(* CODESYS project v35_Linux_Profinet

Project tree, tasks and I/O mapping:
  Device : CODESYS Control for Linux SL, 3S - Smart Software Solutions GmbH, version 4.5.0.0
    application Application
      libraries: Standard, * (System)
      task MainTask (cyclic, interval t#4ms, priority 1) calls PLC_PRG
      task Profinet_CommunicationTask (cyclic, interval t#10ms, priority 14) calls PN_Controller.CommCycle
      task Profinet_IOTask (cyclic, interval t#1ms, priority 1) calls nothing
      program PLC_PRG [ST]
    Ethernet : Ethernet, 3S - Smart Software Solutions GmbH, version 3.5.17.0
        settings: IPAddress = [10,10,2,5]; SubnetMask = [255,255,255,0]; GatewayAddress = [0,0,0,0]; MACAddress = [16#C4,16#00,16#AD,16#8F,16#F7,16#F8]; NetworkInterfaceName = 'X11'; NetworkInterfaceName = "X11"; SaveCommunicationSettings = FALSE
      PN_Controller : PN-Controller, 3S - Smart Software Solutions GmbH, order no. 1, version 4.2.0.0
          settings: Controller Options.IOxSSettings.PSInputDataMapped = True; Controller Options.IOxSSettings.CSOutputDataMapped = True; First IP Address = [10, 10, 2, 10]; Last IP Address = [10, 10, 2, 254]; Default Subnet Mask = [255, 255, 255, 0]; Default Gateway Address = [0, 0, 0, 0]; PDPortDataCheck.PeerStationName = ''
        RIO_Panel1A : 750-375 V02.07.xx (FW 10), WAGO Kontakttechnik GmbH & Co. KG, order no. 750-375, version SW=V02.07.xx (10), HW=01
            settings: Slave parameters.Identification.IP address = [10,10,2,10]; Slave parameters.Identification.Subnet mask = [255,255,255,0]; Slave parameters.Identification.Default gateway = [0,0,0,0]; Slave parameters.Identification.MAC address = [16#00,16#30,16#DE,16#40,16#2C,16#5D]; Slave parameters.Identification.Station name = 'wago.remote.io.2'; Slave parameters.Reduction ratio = 4; PDPortDataCheck.PeerStationName = ''; PDPortDataCheck.PeerStationName = ''
            unmapped channels: Inputs PS, Inputs PS, Inputs PS, Inputs PS
          RIO_Panel1A_S01 : 750-496 8AI 0/4-20 mA s.e., WAGO Kontakttechnik GmbH & Co. KG, order no. 750-496, version SW=V02.07.xx (10), HW=01
              settings: Module parameters.Slot number = 1
            wago_remote_io_2_2_1 : 8AI, INT16[8] I, WAGO Kontakttechnik GmbH & Co. KG, version SW=V02.07.xx (10), HW=01
                settings: 8AI, INT16[8] I.Subslot number = 1; swapInfoInputs = [7,8]
                unmapped channels: Inputs, Inputs PS
          RIO_Panel1A_S02 : 16DO, WAGO Kontakttechnik GmbH & Co. KG, order no. 750-15xx, version SW=V02.07.xx (10), HW=01
              settings: Module parameters.Slot number = 2
            wago_remote_io_2_2_1_1 : 16DO, WAGO Kontakttechnik GmbH & Co. KG, version SW=V02.07.xx (10), HW=01
                settings: 16DO.Subslot number = 1; swapInfoOutputs = [2,2]
                unmapped channels: Digital Outputs .0 - .15, Outputs CS
    SoftMotion General Axis Pool
*)

// Device/Application/PLC_PRG
PROGRAM PLC_PRG
VAR
END_VAR

END_PROGRAM
